Universal Robots PolyScope program: Albert_Samuel_P3.urp

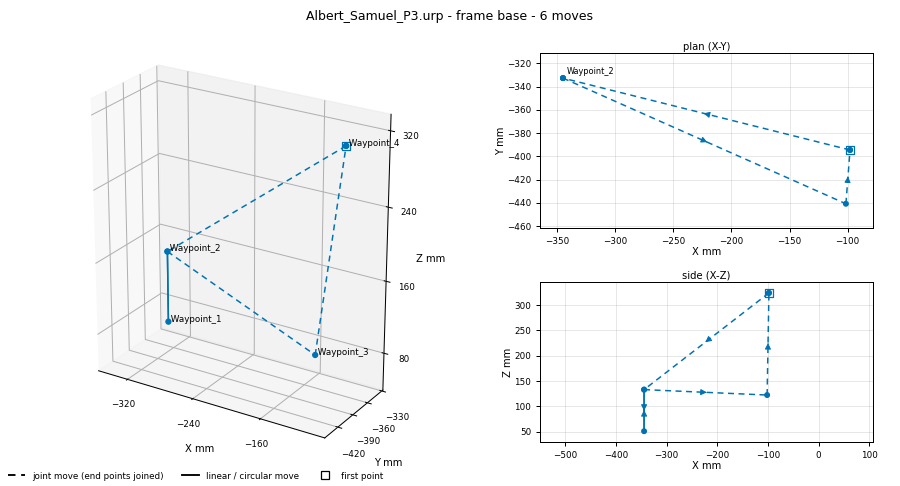
[picture p0: tool path of Albert_Samuel_P3.urp in frame base, 6 of 6 moves have a stored position in this frame; points joined in program order, loops and branches not executed]
Program Albert_Samuel_P3 (installation=default directory=/programs createdIn=5.14.5 lastSavedIn=5.14.5 robotSerialNumber=20195300809)
Calibrated DH parameters: a=[-0.000085, -0.20076, -0.212369, 0.000121, -0.000118, 0]; d=[0.15185, -26.306375, 24.753047, 1.684739, 0.085386, 0.092088]; alpha=[1.572149, -0.00522, -0.011864, 1.571339, -1.571085, 0]; deltaTheta=[0, 0.599885, -0.513355, -0.086555, 0.000006, 0]
InitVariablesNode
Robot Program (runOnlyOnce=false)
  MoveJ speed 60 deg/s, acceleration 80 deg/s^2 (useActiveTCP=true) feature=Base
    Waypoint Waypoint_4: TCP in base x=-97.99 y=-394.459 z=324.162 mm, rx=2.2311 ry=0.1427 rz=-0.0075 rad; joints [-83.374, -68.189, -99.755, -50.174, 86.77, -182.099] deg; TCP offset x=0 y=0 z=174 mm, rx=0 ry=0 rz=0 rad
    URCap Gripper (Robotiq_Grippers, Robotiq Inc.) dataModel(position=0.0, force=0.0, positionInDouble=0.0, forceInDouble=0.0, blocking=true, slaveIds=[9], speedInDouble=0.0, speed=0.0)
  MoveJ speed 60 deg/s, acceleration 80 deg/s^2 (useActiveTCP=true) feature=Base
    Waypoint Waypoint_2: TCP in base x=-344.685 y=-332.697 z=133.115 mm, rx=3.0611 ry=-0.0085 rz=0.0846 rad; joints [-123.292, -134.32, -26.373, -107.157, 94.365, -212.301] deg
  MoveL speed 250 mm/s, acceleration 1200 mm/s^2 (useActiveTCP=true) feature=Base
    Waypoint Waypoint_1: TCP in base x=-344.699 y=-332.718 z=50.951 mm, rx=3.061 ry=-0.0085 rz=0.0845 rad; joints [-123.268, -131.006, -54.673, -82.187, 94.329, -212.565] deg
    Wait Sleep waitTime=0.5
    URCap Gripper (Robotiq_Grippers, Robotiq Inc.) dataModel(position=100.0, force=0.0, speed=100.0, positionInDouble=100.0, forceInDouble=0.0, speedInDouble=100.0, slaveIds=[9], blocking=true)
    Wait Sleep waitTime=1
    Waypoint Waypoint_2: TCP in base x=-344.685 y=-332.697 z=133.115 mm, rx=3.0611 ry=-0.0085 rz=0.0846 rad; joints [-123.292, -134.32, -26.373, -107.157, 94.365, -212.301] deg
  MoveJ speed 60 deg/s, acceleration 80 deg/s^2 (useActiveTCP=true) feature=Base
    Waypoint Waypoint_3: TCP in base x=-101.545 y=-440.683 z=122.402 mm, rx=1.9332 ry=-1.8787 rz=0.5296 rad; joints [-84.25, -95.399, -109.079, -34.032, 86.377, -87.007] deg
  Force Frame feature=Plane_good; selection=[1, 1, 0, 0, 0, 0]; wrench=[0, 0, 5, 0, 0, 0]; limitsForce=[0.15, 0.15, 0.15, 1.047198, 1.047198, 1.047198]; limitsMotion=[0.1, 0.1, 0.1, 0.349066, 0.349066, 0.349066]
    Popup Message (haltProgram=false message=Move the robot to the desired position. If the position is correct press OK. inputType=Text)
  Wait Sleep waitTime=0.5
  MoveL speed 70 mm/s, acceleration 1200 mm/s^2 (useActiveTCP=true) feature=Joint_6_name
    MoveDirectionNode (selectedDirection=ZPlus) feature(featureName=Plane_good)
      Until TOOL_CONTACT_DETECTION (allowActions=false retraction=0 decelerationAcceleration=3 decelerationAngularAcceleration=34.906585)
  Force Frame feature=Plane_good; selection=[0, 0, 1, 0, 0, 0]; wrench=[0, 0, 15, 0, 0, 0]; limitsForce=[0.15, 0.15, 0.05, 1.047198, 1.047198, 1.047198]; limitsMotion=[0.1, 0.1, 0.1, 0.349066, 0.349066, 0.349066]
    Wait Sleep waitTime=5
  URCap Gripper (Robotiq_Grippers, Robotiq Inc.) dataModel(position=78.43137254901961, force=0.0, speed=0.0, positionInDouble=78.43137254901961, forceInDouble=0.0, speedInDouble=0.0, slaveIds=[9], blocking=true)
  MoveL speed 70 mm/s, acceleration 1200 mm/s^2 (useActiveTCP=true) feature=Joint_6_name
    MoveDirectionNode (selectedDirection=ZMinus) feature(featureName=Plane_good)
      Until DISTANCE (allowActions=false deceleration=3 distanceNodeType=STOP) Distance=0.05; motionParameters(blendRadius=0)
  Wait Sleep waitTime=1
  MoveJ speed 60 deg/s, acceleration 80 deg/s^2 (useActiveTCP=true) feature=Base
    Waypoint Waypoint_4: TCP in base x=-97.99 y=-394.459 z=324.162 mm, rx=2.2311 ry=0.1427 rz=-0.0075 rad; joints [-83.374, -68.189, -99.755, -50.174, 86.77, -182.099] deg
  Popup Message (haltProgram=false message=Process finished, pick the clothe. inputType=Text)
